Staubli VAL3: ChoosehansPro.pgx

public program ChoosehansPro(num& x_nWorkPlace (dimensions=1), num& x_nProductIndex (dimensions=1), num& x_nMax[] (dimensions=1))
  local num l_nNum
begin
  //  //2013.10.30
  //  //通过数字量来选择产品
  //  //主要用来检测按钮触发
  //  //同工位多产品函数

  //2014.05.30





  //  x_nProductIndex=0
  //  x_nProductIndex=0
  //  l_nNum=0

  if x_nProductIndex>=x_nMax[x_nWorkPlace]
    x_nProductIndex=0
  endIf

  if x_nProductIndex>0
    x_nProductIndex=x_nProductIndex+1
    return

  endIf

  while true
    //工位1
    if dDio["In1_bPrdSta1"]==true and dDio["UsIn_bNull1"]==true and dDio["UsIn_bNull2"]==true
      delay(0.1)
      if dDio["In1_bPrdSta1"]==true and dDio["UsIn_bNull1"]==true and dDio["UsIn_bNull2"]==true
        //
        x_nProductIndex=1
        x_nWorkPlace=1
        return
      endIf
    endIf


    //工位2
    if dDio["In1_bPrdSta2"]==true and dDio["UsIn_bNull3"]==true and dDio["UsIn_bNull3"]==true
      delay(0.1)
      if dDio["In1_bPrdSta2"]==true and dDio["UsIn_bNull3"]==true and dDio["UsIn_bNull4"]==true
        //
        x_nProductIndex=1
        x_nWorkPlace=2
        return
      endIf
    endIf


    //工位3
    if dDio["In1_bPrdSta2"]==true and dDio["UsIn_bNull5"]==true and dDio["UsIn_bNull6"]==true
      delay(0.1)
      if dDio["In1_bPrdSta2"]==true and dDio["UsIn_bNull5"]==true and dDio["UsIn_bNull6"]==true
        //
        x_nProductIndex=1
        x_nWorkPlace=3
        return
      endIf
    endIf







    //2014.06.03
    //*************************************************************************
    //*************************************************************************

    //为大族定制
    //A1,A2,A3,A4
    if dDio["In1_bPrdSta1"]==true and dDio["UsIn_bNull1"]==true and dDio["UsIn_bNull2"]==true
      delay(0.1)
      if dDio["In1_bPrdSta1"]==true and dDio["UsIn_bNull1"]==true and dDio["UsIn_bNull2"]==true
        //
        x_nProductIndex=1
        x_nWorkPlace=1
        x_nMax[1]=4
        return
      endIf
    endIf


    //A1,A2
    if dDio["In1_bPrdSta1"]==true and dDio["UsIn_bNull1"]==true and dDio["UsIn_bNull2"]==true
      delay(0.1)
      if dDio["In1_bPrdSta1"]==true and dDio["UsIn_bNull1"]==true and dDio["UsIn_bNull2"]==true
        //
        x_nProductIndex=1
        x_nWorkPlace=1
        x_nMax[1]=2
        return
      endIf
    endIf

    //A3,A4
    if dDio["In1_bPrdSta1"]==true and dDio["UsIn_bNull1"]==true and dDio["UsIn_bNull2"]==true
      delay(0.1)
      if dDio["In1_bPrdSta1"]==true and dDio["UsIn_bNull1"]==true and dDio["UsIn_bNull2"]==true
        //
        x_nProductIndex=3
        x_nWorkPlace=1
        x_nMax[1]=4
        return
      endIf
    endIf

    //***********************************************************************************
    //**********************************************************************************



    delay(0)
  endWhile




end
